// TIA Portal V20 export
// export: Created 2026-10-03T18:54:34.668872Z, ExportSetting WithDefaults, DisplayName Totally Integrated Automation Portal, DisplayVersion V20 Update 4, DisplayName TIA Portal Openness, DisplayVersion V20 Update 4, DisplayName TIA Portal Version Control Interface, DisplayVersion V20 Update 4, DisplayName SINAMICS Startdrive Advanced, DisplayVersion V20 SP1 Update 1, DisplayName SINAMICS Startdrive G110M, G120, G120C, G120D, G120P, G115D, DisplayVersion V20 SP1 Update 1, DisplayName SINAMICS Startdrive G130, G150, S120, S150, SINAMICS MV, G220, S200, S210, DisplayVersion V20 SP1 Update 1, DisplayName STEP 7 Professional, DisplayVersion V20 Update 4, DisplayName STEP 7 Safety, DisplayVersion V20 Update 2, DisplayName WinCC Basic/Comfort/Advanced, DisplayVersion V20 Update 4, DisplayName WinCC Unified, DisplayVersion V20 Update 4
FUNCTION "SLC_MVM" : Int   // FC21, SCL
TITLE = SLC MVM (masked move)
{ S7_Optimized_Access := 'TRUE' }
VERSION : 0.1
// Replaces MVM Source Mask Dest: the bits of Source where Mask is 1 replace those bits of Dest; the other bits of
//  Dest are kept. Returns the new value of Dest.
// stored: AutoNumber true, IsIECCheckEnabled false, SetENOAutomatically false, UDAEnableTagReadback false
   VAR_INPUT
      Source : Int;   // Value to take the masked bits from
      Mask : Int;   // 1 = take this bit from Source, 0 = keep it from Dest
      Dest : Int;   // Current value of the destination
   END_VAR
BEGIN
   #SLC_MVM := WORD_TO_INT((INT_TO_WORD(#Dest) AND NOT INT_TO_WORD(#Mask)) OR (INT_TO_WORD(#Source) AND INT_TO_WORD(#Mask)));
END_FUNCTION
